{attribute 'qualified_only'}
VAR_GLOBAL
	bCalibrateGyro: BOOL := FALSE;
	bResetGryo: BOOL := FALSE;
END_VAR

(* stored: Version 1.1.0.1, ProductVersion 3.1.4026.18
   GVL GVL_Control: Id {83e9a3cd-fae6-4c81-b962-272ece6f5662} *)
